# EPICS substitutions: IOC/prj/iocBoot/iocLinux/fb_epid.substitutions
# $Id$

file "$(TOP)/prjApp/Db/fb_epid.db"
  {
    {
        P=prj:epid1,
	IN=prj:epid1:sim.VAL,
	OUT=prj:epid1:sim.D,
	MODE=PID,
	CALC=A,
	PERMIT1="prj:epid1:on.VAL",
	PERMIT2="",
	PERMIT3="",
	PERMIT4=""
    }
  }
